Yaskawa INFORM job: DEMONSTRATOR_TEST_EINZELFLAECHE.JBI

/JOB
//NAME DEMONSTRATOR_TEST_EINZELFLAECHE
///FOLDERNAME DEMONSTRATOR
//POS
///NPOS 0,0,0,0,0,0
//ALIAS
///LVARS 0,0,1,0,0,0,0,0
LD000 V_weld
//ARGINFO
///ARGTYPE D,D,D,D,D,D,D,D
///COMMENT
X left
X right
X Offset
Height_left
Height_right
USERFRAME
V_WELD
Kennlinie
//INST
///DATE 2023/01/24 14:22
///ATTR SC,RW
///GROUP1 RB1
///LVARS 1,3,27,0,0,0,0,0
NOP
CALL JOB:SET_ID ARGF33 ARGF"LAGE_NR"
'--------------------------------
'WELD-Geschwindigkeit
CALL JOB:GET_V ARGF40 ARGF"cm/min"
GETS V_weld $RV
CALL JOB:DEMONSTRATOR_A7 ARGF-200000 ARGF200001 ARGF4300 ARGF96000 ARGF96000 ARGF4 ARGFV_weld ARGF8
END
